INTERFACE I_HAL_DO

PROPERTY errId : HAL_ErrorEnum
GET
END_GET
END_PROPERTY

PROPERTY xValue : bool
GET
END_GET
SET
END_SET
END_PROPERTY

END_INTERFACE

(* stored: Version 1.1.0.1, ProductVersion 3.1.4024.6
   Itf I_HAL_DO: Id {91024714-31c5-0650-3137-cca3ae6f3774}
   Property errId: Id {90300fa2-a256-09dc-3624-09027a35ba7c}
   Get Get: Id {7eb76d01-9028-0d44-24b8-237afe51e471}
   Property xValue: Id {55752649-a795-0794-08a4-ae321fd150f7}
   Get Get: Id {15d47da7-4646-0791-3c4d-8c21b3b564bd}
   Set Set: Id {375d98f7-abc5-0f7e-39c7-2a65c1b10b9e} *)
